// TwinCAT 3 PLC project PlcProject1
// ProgramVersion: 3.1.4023.0
// libraries:
//   Tc2_Standard, * (Beckhoff Automation GmbH)
//   Tc2_System, * (Beckhoff Automation GmbH)
//   Tc3_Module, * (Beckhoff Automation GmbH)
//   TcUnit, * (www.tcunit.org)
// project tree:
//   / PlcTask.TcTTO
//   POUs/ MAIN.TcPOU, FB_GatewaySmokeTests.TcPOU
// real-time tasks:
//   TASK PlcTask: cycle T#10ms, priority 20, ADS port 350
//   TASK PlcTask1: cycle T#10ms, priority 21, ADS port 351

CONFIGURATION PlcProject1
    RESOURCE PLC ON TwinCAT3
        TASK PlcTask(INTERVAL := T#10ms, PRIORITY := 20);
        PROGRAM MAIN WITH PlcTask : MAIN;
    END_RESOURCE
END_CONFIGURATION

// ---- POUs/MAIN.TcPOU
PROGRAM MAIN
VAR
    gatewaySmokeTests : FB_GatewaySmokeTests;
END_VAR

TcUnit.RUN();

END_PROGRAM

// ---- POUs/FB_GatewaySmokeTests.TcPOU
FUNCTION_BLOCK FB_GatewaySmokeTests EXTENDS TcUnit.FB_TestSuite

GatewayCanExecuteTcUnit();

METHOD PRIVATE GatewayCanExecuteTcUnit
TEST('GatewayCanExecuteTcUnit');
AssertTrue(
    Condition := TRUE,
    Message := 'Gateway TcUnit smoke test should pass');
TEST_FINISHED();
END_METHOD

END_FUNCTION_BLOCK
